INTERFACE I_VirtualInputSource

METHOD Done : BOOL
END_METHOD

METHOD NextData : BOOL
VAR_INPUT
	nMaxOversampling: UDINT;
END_VAR
END_METHOD

METHOD SourceSync : BOOL
END_METHOD

PROPERTY bEndOfData : BOOL
GET
END_GET
END_PROPERTY

PROPERTY dtTimestamp : DCTIMESTRUCT
GET
END_GET
END_PROPERTY

PROPERTY nContext : DWORD
GET
END_GET
END_PROPERTY

PROPERTY nDataHandle : ULINT
GET
END_GET
END_PROPERTY

PROPERTY tTimestamp : ULINT
GET
END_GET
END_PROPERTY

PROPERTY eSourceState : E_DataSourceState
GET
END_GET
END_PROPERTY

END_INTERFACE

(* stored: Itf I_VirtualInputSource: Id 5824ce83-99b2-4aae-9be2-d0fbb7d17e8a
   Method Done: Id 2e4883e5-aeeb-4e91-91f5-a86928036ea1
   Method NextData: Id 3fd98946-5111-4045-9cee-550261b9970b
   Method SourceSync: Id adc74e4f-e8d5-4f41-ad88-1ba1e193db0a
   Property bEndOfData: Id 04474717-7107-4678-9eb3-e06d92804025
   Get Get: Id 3fdb8170-b9ca-4273-936b-149fb767a2ac
   Property dtTimestamp: Id 2f7a57c8-f996-495e-97a0-3ad33e567167
   Get Get: Id 296fde56-2b43-4430-8a83-bb836705b5e4
   Property nContext: Id 3d89ef11-15f4-473a-8755-8566f4cb8455
   Get Get: Id a4d7b9a8-74db-4db8-91f7-4fceea3ea14e
   Property nDataHandle: Id 6590f30d-7a54-4265-9a94-91668d7a98de
   Get Get: Id e1aabda8-f88b-4141-a124-9f46c5007e06
   Property tTimestamp: Id 036ec1e7-0a14-4816-bdf6-547595fd9060
   Get Get: Id 3127d070-05fe-4797-81d8-74d1c934bbe8
   Property eSourceState: Id 44515c0c-9abc-4996-9d06-947202dee40f
   Get Get: Id bf1845a9-18b0-4677-8e39-973390419006 *)
